TYPE stError :
STRUCT
	code : INT;
	message : STRING(255);
	timestamp : DATE_AND_TIME;
	severity : eSeverity;
END_STRUCT
END_TYPE

(* stored: Version 1.1.0.1, ProductVersion 3.1.4026.18
   DUT stError: Id {c1b2c3d4-1111-1111-1111-111111111111} *)
